PROGRAM IoT_JSON_XML
VAR
	
	//Data Struct and data struct population
	DataValues : IoTDataStruct;
	ReceiveDataValues : IoTDataStruct;
	
	//String send/rec vars
	fb_SendString : FB_MqttCom_String;
	MyRecString: STRING(2000);
	
	//JSON Encoding of Data Struct
	fb_EncodeJSON : FB_JSONEncoding; 
	StringToSend: STRING(2000);
END_VAR

//Populate Data Stuct with data
prgPopulateStructure( DataStructure := DataValues);

//Encode the Data Struct to JSON format
fb_EncodeJSON(DataStruct := DataValues, sJsonDoc2 => StringToSend);

//Send Data Struct as JSON
fb_SendString(sTopicPub:= 'JSON_Data', sPayloadPub:= StringToSend, sTopicSub:= 'JSON_Data', sPayloadRcv => MyRecString);

END_PROGRAM

(* stored: Version 1.1.0.1, ProductVersion 3.1.4024.11
   POU IoT_JSON_XML: Id {86441d78-7a43-41bd-ab52-071d97178c0e}, SpecialFunc None *)
